// LS Electric XG5000 project: parsing_example
// PLC LSPLC_RE
// module base 0 slot 0: 입력 모듈:XBC-EL95A, Input (DC/AC 입력 62점)
// module base 0 slot 1: 출력 모듈:XBC-EL95A, Output (TR/RY 출력 33점)
// module base 0 slot 2: Cnet:XBL-C81A (Cnet 통신 모듈(RS-485))
// module base 0 slot 3: Cnet:XBL-C81A (Cnet 통신 모듈(RS-485))

PROGRAM Interlock (task: 스캔 프로그램)

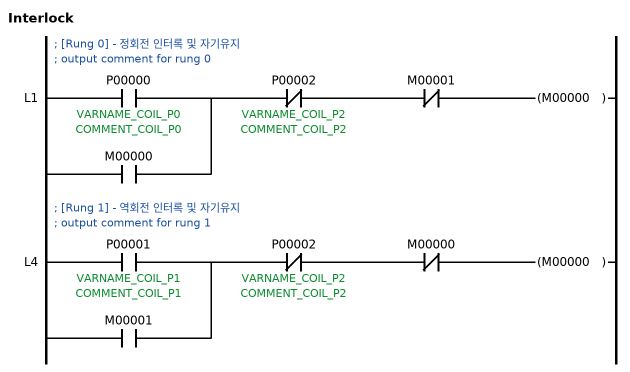
// [Rung 0] - 정회전 인터록 및 자기유지
; L1
LOAD      P00000	// VARNAME_COIL_P0 COMMENT_COIL_P0
OR        M00000
AND NOT   P00002	// VARNAME_COIL_P2 COMMENT_COIL_P2
AND NOT   M00001
OUT       M00000
// output comment: output comment for rung 0
// [Rung 1] - 역회전 인터록 및 자기유지
; L4
LOAD      P00001	// VARNAME_COIL_P1 COMMENT_COIL_P1
OR        M00001
AND NOT   P00002	// VARNAME_COIL_P2 COMMENT_COIL_P2
AND NOT   M00000
OUT       M00000
// output comment: output comment for rung 1

PROGRAM TON_TOF (task: 스캔 프로그램)

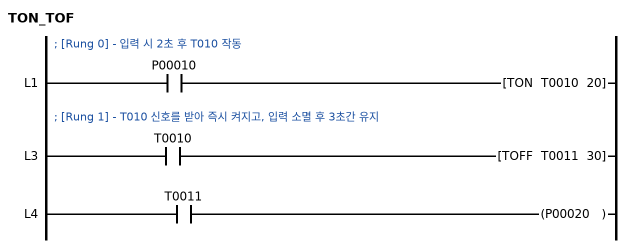
// [Rung 0] - 입력 시 2초 후 T010 작동
; L1
LOAD      P00010
TON       T0010 20
// [Rung 1] - T010 신호를 받아 즉시 켜지고, 입력 소멸 후 3초간 유지
; L3
LOAD      T0010
TOFF      T0011 30
; L4
LOAD      T0011
OUT       P00020

PROGRAM CTU_CTD (task: 스캔 프로그램)

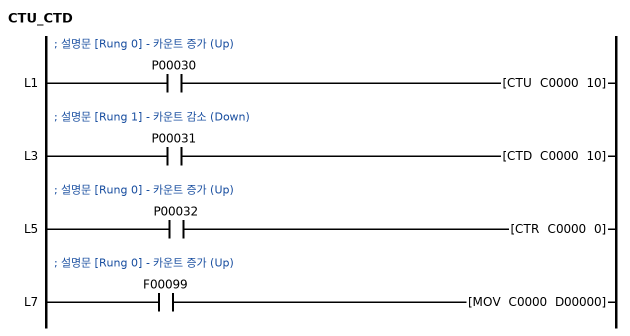
// 설명문 [Rung 0] - 카운트 증가 (Up)
; L1
LOAD      P00030
CTU       C0000 10
// 설명문 [Rung 1] - 카운트 감소 (Down)
; L3
LOAD      P00031
CTD       C0000 10
// 설명문 [Rung 0] - 카운트 증가 (Up)
; L5
LOAD      P00032
CTR       C0000 0
// 설명문 [Rung 0] - 카운트 증가 (Up)
; L7
LOAD      F00099
MOV       C0000 D00000

VARIABLES AND COMMENTS (devices not used above)
P0000A	BIT	VARNAME_COIL_P10
P0000B	BIT	VARNAME_COIL_P11
P0000C	BIT	VARNAME_COIL_P12
P0000D	BIT	VARNAME_COIL_P13
P0000E	BIT	VARNAME_COIL_P14
P0000F	BIT	VARNAME_COIL_P15
P00003	BIT	VARNAME_COIL_P3 // COMMENT_COIL_P3
P00004	BIT	VARNAME_COIL_P4
P00005	BIT	VARNAME_COIL_P5
P00006	BIT	VARNAME_COIL_P6
P00007	BIT	VARNAME_COIL_P7
P00008	BIT	VARNAME_COIL_P8
P00009	BIT	VARNAME_COIL_P9